FUNCTION_BLOCK EL3101
VAR
	_io : EL3xx1_Data;
	{attribute addProperty Name "WcState"}
	_wcState : WcStateInputToggle;
	{attribute addProperty Name "Info data"}
	_infoData : InfoDataAds;
END_VAR

PROPERTY IO : REFERENCE TO EL3xx1_Data
GET
IO REF= _io;
END_GET
END_PROPERTY

PROPERTY WcState : REFERENCE TO WcStateInputToggle
GET
WcState REF= _wcState;
END_GET
END_PROPERTY

END_FUNCTION_BLOCK

(* stored: Version 1.1.0.1, ProductVersion 3.1.4024.9
   POU EL3101: Id {fc0415c9-364c-00ab-35b5-a8cf5e8e4e23}, SpecialFunc None
   Property IO: Id {ee8b370b-96d9-085a-1eaa-9fa334b0f0c5}
   Get Get: Id {f59c4bdb-bb4b-09c2-198d-a09ce91a38e3}
   Property WcState: Id {e91af986-d7ff-0238-31b5-a0ee99bea7ca}
   Get Get: Id {e2b6010e-2ba3-0f9c-2181-79caa63bcac0} *)
